// TIA Portal V19 export
FUNCTION_BLOCK "Deckel"   // FB1190, LAD
TITLE = Deckelsteuerung
{ S7_Optimized_Access := 'TRUE' }
// stored: AutoNumber false, MemoryReserve 100, SetENOAutomatically true
   VAR
      In { ExternalAccessible := 'False'; ExternalVisible := 'False'; ExternalWritable := 'False'} : Struct
         NotHalt : Bool;
         Si_24VDC_links : Bool;
         Si_24VDC_rechts : Bool;
         Auto : Bool;
         Hand : Bool;
         Tipp : Bool;
         ErrQ : Bool;
         T_links_auf : Bool;   // Paneltaste
         T_links_zu : Bool;   // Paneltaste
         T_rechts_auf : Bool;   // Paneltaste
         T_rechts_zu : Bool;   // Paneltaste
         SRM_links_auf : Bool;
         SRM_links_zu : Bool;
         SRM_rechts_auf : Bool;
         SRM_rechts_zu : Bool;
         S_links_auf : Bool;
         S_links_zu : Bool;
         S_rechts_auf : Bool;
         S_rechts_zu : Bool;
      END_STRUCT;
   END_VAR
   VAR RETAIN
      Param { ExternalAccessible := 'False'; ExternalVisible := 'False'; ExternalWritable := 'False'} : Struct
         "TO" : Time := T#27s;
         gleichzeitig : Time := T#1s500ms;
      END_STRUCT;
      Zst { ExternalAccessible := 'False'; ExternalVisible := 'False'; ExternalWritable := 'False'} : Struct
         Fehler : Bool;
         Sperre_Pos_li : Bool;
         Sperre_Pos_re : Bool;
         Req_links_auf : Bool;
         Req_rechts_auf : Bool;
         TW_sicher : Bool;
         Ist_Pos_links : Int;   // 0% = auf; 100% = zu
         Ist_Pos_rechts : Int;   // 0% = auf; 100% = zu
      END_STRUCT;
      Out { ExternalAccessible := 'False'; ExternalVisible := 'False'; ExternalWritable := 'False'} : Struct
         links_auf : Bool;
         links_zu : Bool;
         rechts_auf : Bool;
         rechts_zu : Bool;
      END_STRUCT;
      Mld { ExternalAccessible := 'False'; ExternalVisible := 'False'; ExternalWritable := 'False'} : Struct
         TO_links_auf : Bool;
         TO_links_zu : Bool;
         TO_rechts_auf : Bool;
         TO_rechts_zu : Bool;
         Si_24VDC_links : Bool;
         Si_24VDC_rechts : Bool;
         n_Auto : Bool;
         SF_gleich_li_auf : Bool;
         SF_gleich_li_zu : Bool;
         SF_gleich_re_auf : Bool;
         SF_gleich_re_zu : Bool;
      END_STRUCT;
   END_VAR
   VAR
      IEC_Timer { ExternalAccessible := 'False'; ExternalVisible := 'False'; ExternalWritable := 'False'} : Struct
         TO_li_auf { S7_SetPoint := 'True'} : TON_TIME;
         TO_li_zu { S7_SetPoint := 'True'} : TON_TIME;
         TO_re_auf { S7_SetPoint := 'True'} : TON_TIME;
         TO_re_zu { S7_SetPoint := 'True'} : TON_TIME;
         gleich_li_auf { S7_SetPoint := 'True'} : TON_TIME;
         gleich_li_zu { S7_SetPoint := 'True'} : TON_TIME;
         gleich_re_auf { S7_SetPoint := 'True'} : TON_TIME;
         gleich_re_zu { S7_SetPoint := 'True'} : TON_TIME;
      END_STRUCT;
   END_VAR
   VAR_TEMP
      TO_links_auf : Bool;
      TO_links_zu : Bool;
      TO_rechts_auf : Bool;
      TO_rechts_zu : Bool;
   END_VAR
BEGIN

REGION Network 1 (SCL): Input / Sammelstörung
   // Panelbedienung und Sensoren --> Input()
   // Not-Halt
   #In.NotHalt :=  NOT "DB_PNOZ_IN_Out".In.NH_Frg_Deckel;

   IF #In.ErrQ THEN
       #Zst.Fehler := FALSE;
   END_IF;

   IF #In.NotHalt OR NOT #In.Si_24VDC_links OR NOT #In.Si_24VDC_rechts OR #Mld.TO_links_auf OR #Mld.TO_links_zu
       OR #Mld.TO_rechts_auf OR #Mld.TO_rechts_zu
   THEN
       #Zst.Fehler := TRUE;
   END_IF;
END_REGION

REGION Network 2 (SCL): Ansteuerung
   IF NOT #Zst.Fehler THEN
       IF #In.Auto AND #Zst.TW_sicher THEN // Automatikbetrieb
           // Linke Seite
           #Out.links_auf := #Zst.Req_links_auf;
           #Out.links_zu := NOT #Zst.Req_links_auf;
           // Rechte Seite
           #Out.rechts_auf := #Zst.Req_rechts_auf;
           #Out.rechts_zu := NOT #Zst.Req_rechts_auf;

       ELSIF #In.Hand AND #Zst.TW_sicher THEN // Handbetrieb
           // Linke Seite
           IF #In.T_links_auf AND NOT #In.T_links_zu THEN
               #Out.links_auf := TRUE;
               #Out.links_zu := FALSE;
           END_IF;
           IF #In.T_links_zu AND NOT #In.T_links_auf THEN
               #Out.links_zu := TRUE;
               #Out.links_auf := FALSE;
           END_IF;
           // Rechte Seite
           IF #In.T_rechts_auf AND NOT #In.T_rechts_zu THEN
               #Out.rechts_auf := TRUE;
               #Out.rechts_zu := FALSE;
           END_IF;
           IF #In.T_rechts_zu AND NOT #In.T_rechts_auf THEN
               #Out.rechts_zu := TRUE;
               #Out.rechts_auf := FALSE;
           END_IF;
       ELSIF #In.Tipp THEN  // Tippbetrieb
           // Linke Seite
           #Out.links_auf := #In.T_links_auf AND NOT #In.T_links_zu;
           #Out.links_zu := #In.T_links_zu AND NOT #In.T_links_auf AND #Zst.TW_sicher;

           // Rechte Seite
           #Out.rechts_auf := #In.T_rechts_auf AND NOT #In.T_rechts_zu;
           #Out.rechts_zu := #In.T_rechts_zu AND NOT #In.T_rechts_auf AND #Zst.TW_sicher;
       ELSE
           #Out.links_auf := FALSE;
           #Out.links_zu := FALSE;
           #Out.rechts_auf := FALSE;
           #Out.rechts_zu := FALSE;
       END_IF;

   ELSE // Not-Halt
       #Out.links_auf := FALSE;
       #Out.links_zu := FALSE;
       #Out.rechts_auf := FALSE;
       #Out.rechts_zu := FALSE;
   END_IF;

   // Endlagen erreicht
   IF #In.S_links_auf OR #In.SRM_links_auf THEN
       #Out.links_auf := FALSE;
   END_IF;
   IF #In.S_links_zu OR #In.SRM_links_zu THEN
       #Out.links_zu := FALSE;
   END_IF;
   IF #In.S_rechts_auf OR #In.SRM_rechts_auf THEN
       #Out.rechts_auf := FALSE;
   END_IF;
   IF #In.S_rechts_zu OR #In.SRM_rechts_zu THEN
       #Out.rechts_zu := FALSE;
   END_IF;


   REGION Ist-Position
       // Ist-Pos simulieren für Visu 
       IF #Out.links_auf AND "Imp_10Hz" AND NOT #In.S_links_auf THEN
           #Zst.Ist_Pos_links := MAX(IN1 := 5, IN2 := (#Zst.Ist_Pos_links - 1));
       ELSIF #In.S_links_auf THEN
           #Zst.Ist_Pos_links := 0;
       END_IF;

       IF #Out.rechts_auf AND "Imp_10Hz" AND NOT #In.S_rechts_auf THEN
           #Zst.Ist_Pos_rechts := MAX(IN1 := 5, IN2 := (#Zst.Ist_Pos_rechts - 1));
       ELSIF #In.S_rechts_auf THEN
           #Zst.Ist_Pos_rechts := 0;
       END_IF;

       // Ist-Pos simulieren für Visu 
       IF #Out.links_zu AND "Imp_5Hz" AND NOT #In.S_links_zu THEN
           #Zst.Ist_Pos_links := MIN(IN1 := 95, IN2 := (#Zst.Ist_Pos_links + 1));
       ELSIF #In.S_links_zu THEN
           #Zst.Ist_Pos_links := 100;
       END_IF;

       IF #Out.rechts_zu AND "Imp_5Hz" AND NOT #In.S_rechts_zu THEN
           #Zst.Ist_Pos_rechts := MIN(IN1 := 95, IN2 := (#Zst.Ist_Pos_rechts + 1));
       ELSIF #In.S_rechts_zu THEN
           #Zst.Ist_Pos_rechts := 100;
       END_IF;
   END_REGION
END_REGION

REGION Network 3 (SCL): Possperre
   // Überfahren verboten
   #Zst.Sperre_Pos_li := NOT (#In.S_links_auf XOR #In.S_links_zu)  OR #Out.links_auf OR #Out.links_zu;

   #Zst.Sperre_Pos_re := NOT (#In.S_rechts_auf XOR #In.S_rechts_zu) OR #Out.rechts_auf OR #Out.rechts_zu;
END_REGION

REGION Network 4 (SCL): Überwachung / Alarme
   // Sicherungsfall / Zeitüberschreitung
   // Sicherungsfall 24V DC links
   #Mld.Si_24VDC_links := NOT #In.Si_24VDC_links AND NOT #In.NotHalt;
   // Sicherungsfall 24V DC rechts
   #Mld.Si_24VDC_rechts := NOT #In.Si_24VDC_rechts AND NOT #In.NotHalt;

   // nicht in Automatik
   #Mld.n_Auto := NOT #In.Auto AND "DB_ANLAGE".BA.Automat_ein;

   // Zeitüberschreitung links öffnen
   #IEC_Timer.TO_li_auf(IN := #Out.links_auf AND NOT #In.S_links_auf,
                        PT := #Param.TO,
                        Q => #TO_links_auf);
   IF #TO_links_auf THEN
       #Mld.TO_links_auf := TRUE;
   ELSIF #In.ErrQ THEN
       #Mld.TO_links_auf := FALSE;
   END_IF;
   // Zeitüberschreitung links schließen
   #IEC_Timer.TO_li_zu(IN := #Out.links_zu AND NOT #In.S_links_zu,
                        PT := #Param.TO,
                        Q => #TO_links_zu);
    IF #TO_links_zu THEN
        #Mld.TO_links_zu := TRUE;
    ELSIF #In.ErrQ THEN
        #Mld.TO_links_zu := FALSE;
    END_IF;
     // Zeitüberschreitung rechts öffnen
    #IEC_Timer.TO_re_auf(IN := #Out.rechts_auf AND NOT #In.S_rechts_auf,
                         PT := #Param.TO,
                         Q => #TO_rechts_auf);
    IF #TO_rechts_auf THEN
        #Mld.TO_rechts_auf := TRUE;
    ELSIF #In.ErrQ THEN
        #Mld.TO_rechts_auf := FALSE;
    END_IF;
    // Zeitüberschreitung rechts schließen
    #IEC_Timer.TO_re_zu(IN := #Out.rechts_zu AND NOT #In.S_rechts_zu,
                        PT := #Param.TO,
                        Q => #TO_rechts_zu);
    IF #TO_rechts_zu THEN
        #Mld.TO_rechts_zu := TRUE;
    ELSIF #In.ErrQ THEN
        #Mld.TO_rechts_zu := FALSE;
    END_IF;
   // Sensor und SRM Zylinder Zeitfenster überwachen 
    #IEC_Timer.gleich_li_auf(IN := #In.SRM_links_auf AND NOT #In.S_links_auf,
                             PT := #Param.gleichzeitig,
                             Q => #Mld.SF_gleich_li_auf);
    // Sensor und SRM Zylinder Zeitfenster überwachen 
    #IEC_Timer.gleich_li_zu(IN := #In.SRM_links_zu AND NOT #In.S_links_zu,
                             PT := #Param.gleichzeitig,
                             Q => #Mld.SF_gleich_li_zu);
     // Sensor und SRM Zylinder Zeitfenster überwachen 
     #IEC_Timer.gleich_re_auf(IN := #In.SRM_rechts_auf AND NOT #In.S_rechts_auf,
                             PT := #Param.gleichzeitig,
                             Q => #Mld.SF_gleich_re_auf);
    // Sensor und SRM Zylinder Zeitfenster überwachen 
    #IEC_Timer.gleich_re_zu(IN := #In.SRM_rechts_zu AND NOT #In.S_rechts_zu,
                            PT := #Param.gleichzeitig,
                            Q => #Mld.SF_gleich_re_zu);
END_REGION
END_FUNCTION_BLOCK
